TYPE ST_Recipe_UBF_PARAM :
STRUCT
	(******BottleSupplySorter********)	
(*******************************BottleSupplySorter Product Type**************************************************************************)	
	//Sorter butelek, typ produktu
	iBottleSorterProductTypeShow												:	ST_DIParametrr;					// 		Typ produktu
	uiBottleSorterIndexShow														:	ST_DIParametrr;					// 		Index butelki 	
	                                                                   
(*******************************BottleSupplySorterHopperTransporter**************************************************************************)	
	//Sorter butelek, transporter zasobnika
	bBottleSorterHopperTransporterEnableShow									:	ST_BoolParametr;					//  	Aktywacja
	iBottleSorterHopperConveyorRunningSpeedSVShow								:	ST_DIParametrr;	//:= 5;			// 		Prędkość | [%] (1-100)
	iBottleSorterHopperConveyorEmptyingSpeedSVShow								:	ST_DIParametrr;	//:= 7;			// 		Prędkość, opróżnianie	| [%] (1-100)
	iBottleSorterDistanceToFindElementOnTransferConveyorLimitRunningSVShow		:	ST_DIParametrr;	//:= 610; 		// 		Odległość do butelek | [mm] (10-10_000)                                  		
	iBottleSorterDistanceToFindElementOnTransferConveyorLimitEmptyingSVShow		:	ST_DIParametrr;	//:= 500; 		// 		Odległość do butelek - opróżnianie | [mm] (10-10_000)                                       		

(*******************************BottleSupplySorterTransferTransporter**************************************************************************)
	//Sorter butelek, transporter transferowy	
	bBottleSorterTransferTransporterEnableShow									:	ST_BoolParametr;					// 		Aktywacja
	iBottleSorterTransferConveyorRunningSpeedSVShow								:	ST_DIParametrr;	//:= 5;			// 		Prędkość | [%] (1-100)	
	iBottleSorterTransferConveyorEmptyingSpeedSVShow							:	ST_DIParametrr;	//:= 7;			// 		Prędkość, opróżnianie | [%] (1-100)
	iBottleSorterDistanceToFindElementOnSupplyConveyorDownstairsLimitSVShow		:	ST_DIParametrr;	//:= 600;			// 		Odległość do butelek - stop zasypu | [mm] (10-10_000)
                                                                               
(*******************************BottleSupplySorterSupplyTransporter**************************************************************************)	
	//Sorter butelek, transporter zasypowy
	bBottleSorterSupplyTransporterEnableShow									:	ST_BoolParametr;					// [H] 	Aktywacja
	uiBottleSorterSupplyTransporterRunningSpeedSVShow							:	ST_UdiParametr;		//:= 1_000;		// 		Prędkość | [obr/min] (10-10_000)	
	uiBottleSorterSupplyTransporterEmptingSpeedSVShow							:	ST_UdiParametr;		//:= 1_000;		// 		Prędkość, opróżnianie | [obr/min] (10-10_000)                                                                   
	lrBottleSorterModuloMoveOffsetSVShow										:   ST_LrParametr;				// 		Kat sprawdzania | [°] (1-360)	                                                                            
	//Logika zasypu - warunek pierwszy	                                                            
	iBottleSorterSensorsCountFirstConditionSVShow								:	ST_DIParametrr;					// 		Limit butelek
	iBottleSorterSupplyTimeFirstConditionSVShow									:	ST_DIParametrr;					// 		Czas zasypu | [ms] (10-10_000)                                                                                                    		
	//Logika zasypu - warunek drugi	 	                                                                                       		
	iBottleSorterSensorsCountSecondConditionMinSVShow							:	ST_DIParametrr;					// 		Limit butelek, min
	iBottleSorterSensorsCountSecondConditionMaxSVShow							:	ST_DIParametrr;					// 		Limit butelek, max
	iBottleSorterSupplyTimeSecondConditionSVShow								:	ST_DIParametrr;					// 		Czas zasypu | [ms] (10-10_000)                                                                                                  		
	//Logika zasypu - warunek trzeci 	                                                                                       		
	iBottleSorterSensorsCountThirdConditionSVShow								:	ST_DIParametrr;					// 		Limit butelek
	iBottleSorterSupplyTimeThirdConditionSVShow									:	ST_DIParametrr;					// 		Czas zasypu | [ms] (10-10_000)
	                                                                            	
(*******************************BottleSupplySorterWheel**************************************************************************)	
	//Sorter butelek, Stól
	bBottleSorterWeelEnableShow													:	ST_BoolParametr;					// [H]	Aktywacja
	lrBottleSorterWheelSpeedSVShow												:   ST_LrParametr; //:= 20;			// 		Prędkość | [obr/min] (5-100)	            
	lrBottleSorterWheelEmptyingSpeedSVShow										:   ST_LrParametr; //:= 30;			// 		Prędkość, opróżnianie | [obr/min] (5-100)	
		
(*******************************BottleSupplySorterBrush**************************************************************************)		
	//Sorter butelek, szczotka
	bBottleSorterBrushEnableShow												:	ST_BoolParametr;					//		Aktywacja
	lrBottleSorterBrushHeightPositionSVShow										:   ST_LrParametr; // := 71;			// 		Wysokosc | [mm] (10-200)	
	iBottleSorterBrushRunningSpeedSVShow										:	ST_DIParametrr; 		 			// 		Prędkość | [%] (1-100)	            
	iBottleSorterBrushEmptyingSpeedSVShow										:	ST_DIParametrr; 		 			// 		Prędkość, opróżnianie | [%] (1-100)                                                              		         	
	
(*********************************BottleSupplyRobot*******************************************************************)

	//Sorter butelek, robot
	bBottleSorterRobotEnableShow												:	ST_BoolParametr;					// 		Aktywacja     
	nBottleSorterRobotRecipeId													:	ST_UdiParametr;					//		Nr receptury                                                                   
	//Czasy przyssania i oddmuchu                                                                                                                              
	lrBottleSorterRemainingTimeToSuctionShow             						:   ST_LrParametr;				// 		Wyprzedzenie przyssania | [ms] (0-200)
	lrBottleSorterSuckerSuctionTimeShow											:   ST_LrParametr;				// 		Czas przyssania	| [ms] (10-1000)
    lrBottleSorterRemainingTimeToRejectShow             						:   ST_LrParametr;				// 		Wuprzedzenie oddmuchu | [ms] (0-200)
	lrBottleSorterEjectorPulseShow                                       		:   ST_LrParametr;				// 		Czas oddmuchu	| [ms] (10-1000)			                                                                                                    		                                                                                                        		
	//Pkt. poboru i dokładania                                                                                 		                                                                                                          		
	lrBottleSorterZPickAboveTheBottleSVShow										:   ST_LrParametr;				// 		Wysokość pobierania butelki
	lrBottleSorterZPickMoveSVShow												:   ST_LrParametr;				// 		Odległość zjazdu w dół łapanie butelki 	                                                                                               	   		                                                                                     		
	lrBottleSorterSafetyHeightSVShow											:   ST_LrParametr;	//:= 150;  		// 		Wysokość obracania chwytaka | [mm] (0-1000)

(*********************************BottleReciever*******************************************************************)

	//Sorter butelek, robot
	bBottleSorterRecieverEnableShow												:	ST_BoolParametr;					// 		Aktywacja   
	bBottleSorterRecieverSlot1EnableShow										:	ST_BoolParametr;					// 		Aktywacja  
	bBottleSorterRecieverSlot2EnableShow										:	ST_BoolParametr;				// 		Aktywacja  
	bBottleSorterRecieverSlot3EnableShow										:	ST_BoolParametr;					// 		Aktywacja  
	lrBottleSorterRecieverHeightPositionSVShow									:   ST_LrParametr;				// 		Wysokosc | [mm] (10-200)	

END_STRUCT
END_TYPE

(* stored: Version 1.2.0.0, ProductVersion 3.1.4026.13, FileIdentifier 0057a3d0c5a7b722dee6f98bd6ae3db4142bec1d, FileSignature 87faaaa6a326edbf51ef9ce85b9e210ac01c4bc4fb1de1dc2e8d0a8e1c0548f96c7ed57414089e525b1364643f4d5a43f1c6633fa72fd5fbb33c104b457490d2b8a86b104cdee2a52c54d4c8e4857f5023eed778a143bb9b3124c38f95773145cbd78185f0cd1297e407f0ba53ef77595c6d61adea22f2deb5da8f103492510513e022835bc186cc96f45a40cc057987e2f0e60afe1e0de6a5f0fa8dd87d141a7491c03c22c5fc871264137be31fe165fab3b0dcd4204ec879b3376dc111c6a964c710f6ff1eedf4337fe73d04cb1794791edd90b2166c72f315712a933cc5d085bf9b3ecdf96f12e30bcbf17749f7807a98570e57329a3f3d4109291455624c
   DUT ST_Recipe_UBF_PARAM: Id {52c6428d-c5a9-4ecd-8d97-b3e9abc10d59} *)
